# B&R Automation Studio project A2019059_Linka_Power_CP (part 60)

#### Main.st - Init, cyclic, exit code
```iecst
PROGRAM _INIT
	(* Insert code here *)

END_PROGRAM

PROGRAM _CYCLIC

	//Alarmy pracoviska č.1 (100 - 199)//
	//A100 - ST1_Vytah - paletka na vystupe dopravnika vytahu !!!
	//A101 - ST1_Vytah - narusenie optickej bariery !!!
	//A102 - ST1_Vytah - porucha navezenia paletky na dopravnik vytahu !!!
	//A103 - ST1_Vytah - porucha precitania kodu paletky !!!
	//A104 - ST1_Vytah - porucha komunikacie zo serverom !!!
	//A105 - ST1_Vytah - porucha odoslania fotiek na server !!!
	//A106 - ST1_Vytah - CAM 2 porucha komunikacie FTP !!!
	//A107 - ST1_Vytah - CAM 3 porucha komunikacie FTP !!!
	//A108 - ST1_Vytah - CAM 4 porucha komunikacie FTP !!!
	//A109 - ST1_Vytah - CAM 5 porucha komunikacie FTP !!!
	//A110 - ST1_Vytah - porucha serva zdvihu vytahu !!!
	//A111 - ST2_Srobovanie - porucha vysunutia centrovacky !!!
	//A112 - ST2_Srobovanie - porucha zasunutia centrovacky !!!
	//A113 - ST2_Srobovanie - porucha precitania kodu paletky !!!
	//A114 - ST2_Srobovanie - porucha komunikacie zo serverom !!!
	//A115 - ST2_Srobovanie - porucha odoslania fotiek na server !!!
	//A116 - ST2_Srobovanie - CAM 6 porucha komunikacie FTP !!!
	//A117 - ST2_Srobovanie - porucha serva manipulatora os X !!!
	//A118 - ST2_Srobovanie - porucha serva manipulatora os Y !!!
	//A119 - ST2_Srobovanie - skrutka K30 nieje pripravena !!!
	//A120 - ST2_Srobovanie - skrutka M5 nieje pripravena !!!
    //A121 - ST2_Srobovanie - skrutka M4 nieje pripravena !!!
    //A122 - P1_Robot - porucha napajania !!!
    //A123 - P1_Robot - nieje online !!!
    //A124 - Pracovisko 1 - Porucha tlaku vzduchu !!!
    //A125 - Pracovisko 1 - Modul DI11 nieje online !!!
    //A126 - Pracovisko 1 - Modul DI12 nieje online !!!
    //A127 - Pracovisko 1 - Modul DI13 nieje online !!!
    //A128 - Pracovisko 1 - Modul DI14 nieje online !!!
    //A129 - Pracovisko 1 - Modul DM11 nieje online !!!
    //A130 - Pracovisko 1 - Modul DS11 nieje online !!!
	//A131 - Pracovisko 1 - Modul DS12 nieje online !!!
	//A132 - Pracovisko 1 - Modul SI11 nieje online !!!
	//A133 - Pracovisko 1 - Modul SI12 nieje online !!!
    //A134 - Pracovisko 1 - Ventilovy termnal VT4 nieje online !!!
    //A135 - Pracovisko 1 - Ventilovy termnal VT5 nieje online !!!
    //A136 - ST2_Srobovanie - Skrutkovacka K30 nieje online !!!
    //A137 - ST2_Srobovanie - Skrutkovacka M5 nieje online !!!
    //A138 - ST2_Srobovanie - Skrutkovacka M4 nieje online !!!
    //A139 - Pracovisko 1 - Kamery KAM2, KAM4 a KAM6 niesu online !!!
    //A140 - Pracovisko 1 - Kamera KAM3 nieje online !!!
	//A141 - Pracovisko 1 - Kamera KAM5 nieje online !!!
    //A142 - ST2_Srobovanie - Porucha vysunutia skrutkovacky K30 !!!
    //A143 - ST2_Srobovanie - Porucha vysunutia skrutkovacky M5  !!!
    //A144 - ST2_Srobovanie - Porucha vysunutia skrutkovacky M4 !!!
	//A145 - P1_Robot - porucha !!!
    //A146 - ST2_Srobovanie - Presiahnuty cas skrutkovania skrutky K30 !!!
    //A147 - ST2_Srobovanie - Presiahnuty cas skrutkovania skrutky M5 !!!
    //A148 - ST2_Srobovanie - Presiahnuty cas skrutkovania skrutky M4 !!!
    //A149 - ST2_Srobovanie - Skrutkovacka K30 nieje READY !!!
    //A150 - ST2_Srobovanie - Skrutkovacka M5 nieje READY !!!
    //A151 - ST2_Srobovanie - Skrutkovacka M4 nieje READY !!!
    //A152 - Pracovisko 1 - Prekrocena teplota motora vrchneho dopravnika !!!
    //A153 - Pracovisko 1 - Prekrocena teplota motora spodneho dopravnika !!!
    //A154 - Pracovisko 1 - Narusenie optickej bariery na vstupe !!!
    //A155 - ST1_Vytah - Prekrocena teplota motora dopravnika !!!
    //A156 - Pracovisko 1 - Bolo stlacene tlacitko CS na ovladacom paneli !!!
    //A157 - Pracovisko 1 - Bolo stlacene tlacitko CS na rozvodnej skrini !!!
    //A158 - Pracovisko 1 - Bolo stlacene tlacitko CS robota !!!
    //A159 - P1_Robot - Porucha odobratia foamov z paletky !!!
    //A160 - P1_Robot - Porucha odobratia busbarov z paletky !!!
    //A161 - ST2_Srobovanie - Porucha vyvezenia paletky zo stopra !!!
    //A162 - P1_Akumulacny stoper - Porucha vyvezenia paletky zo stopra !!!
    //A163 - P1_Spodny stoper - Porucha vyvezenia paletky zo stopra !!!
    //A164 - ST1_Vytah - Porucha komunikacie s kamerou CAM 2 !!!
    //A165 - ST1_Vytah - Porucha komunikacie s kamerou CAM 5 !!!
    //A166 - ST1_Vytah - Porucha komunikacie s kamerou CAM 4 !!!
    //A167 - ST1_Vytah - Porucha komunikacie s kamerou CAM 3 !!!
    //A168 - ST2_Srobovanie - Porucha komunikacie s kamerou CAM 6 !!!

	//******************************Configurácia alarmov**************************************//
    MpAlarmXCore_1.Enable:= TRUE;
    MpAlarmXCore_1.MpLink:= ADR(gAlarmXCore);
    MpAlarmXCore_1();

    //*****************************Configurácia histórie alarmov*****************************//

    MpAlarmXHistory_1.Enable:= TRUE;
    MpAlarmXHistory_1.MpLink:= ADR(gAlarmXHistory);
    MpAlarmXHistory_1.DeviceName:= ADR('HDD_AlarmHistory');
    MpAlarmXHistory_1();

    //****************************Archivácia alarmov na disk PLC******************************//
    IF P1_AlarmyVizu.ArchivaciaAlarmov THEN
        MpAlarmXHistory_1.Export:= TRUE;
        P1_AlarmyVizu.ArchivaciaAlarmov:= FALSE;
    ELSIF P2_AlarmyVizu.ArchivaciaAlarmov THEN
        MpAlarmXHistory_1.Export:= TRUE;
        P2_AlarmyVizu.ArchivaciaAlarmov:= FALSE;
    ELSIF P34_AlarmyVizu.ArchivaciaAlarmov THEN
        MpAlarmXHistory_1.Export:= TRUE;
        P34_AlarmyVizu.ArchivaciaAlarmov:= FALSE;
    END_IF

    IF MpAlarmXHistory_1.Error THEN
        MpAlarmXHistory_1.Export:= FALSE;
    ELSIF MpAlarmXHistory_1.CommandDone THEN
        MpAlarmXHistory_1.Export:= FALSE;
    END_IF

    //***********************************Príznak pracovisko 1 stav PORUCHA*****************************************//

    FOR a:=100 TO 199 BY 1 DO
        P1_Alarmy[a];
        IF P1_Alarmy[a] = TRUE THEN
            P1_Pracovisko.STAV.PORUCHA:= TRUE;
        END_IF
    END_FOR

    //**********************************Porucha tlaku vzduchu*********************************************************//
    IF CasKontroly_TlakVzduchu.Q THEN
        P1_Alarmy[124]:= TRUE;
        P1_PoruchaST1:= TRUE;
        P1_PoruchaST2:= TRUE;
    END_IF

    IF Safety.STAV.P1_ZonaBunky_AKTIVNA AND NOT P1_Pracovisko.IN.PrivodVzduchu_SnimacTlaku_S18 THEN
        CasKontroly_TlakVzduchu.IN:= TRUE;
    ELSE
        CasKontroly_TlakVzduchu.IN:= FALSE;
    END_IF

    CasKontroly_TlakVzduchu.PT:= T#10s;
    CasKontroly_TlakVzduchu();

    //**********************************Porucha - kamerovy systém nieje online****************************************//
    IF CasKontroly_KAMsystem.Q THEN
        IF NOT Linka.STAV.WenglorControlUnit_OK THEN
            P1_Alarmy[149]:= TRUE;
            P1_PoruchaST1:= TRUE;
            P1_PoruchaST2:= TRUE;
        END_IF
        IF NOT CAM3.STAV.READY THEN
            P1_Alarmy[140]:= TRUE;
            P1_PoruchaST1:= TRUE;
            P1_PoruchaST2:= TRUE;
        END_IF
        IF NOT CAM5.STAV.READY THEN
            P1_Alarmy[141]:= TRUE;
            P1_PoruchaST1:= TRUE;
            P1_PoruchaST2:= TRUE;
        END_IF
    END_IF

    IF Safety.STAV.P1_ZonaBunky_AKTIVNA AND NOT P1_Pracovisko.STAV.Kamery_OK THEN
        CasKontroly_KAMsystem.IN:= TRUE;
    ELSE
        CasKontroly_KAMsystem.IN:= FALSE;
    END_IF

    CasKontroly_KAMsystem.PT:= T#2s;
    CasKontroly_KAMsystem();

    //**********************************Porucha - moduly niesu online**************************************************//
    IF CasKontroly_Moduly.Q THEN
        IF NOT P1_Pracovisko.STAV.ModulDI11_OK THEN
            P1_Alarmy[125]:= TRUE;
            P1_PoruchaST1:= TRUE;
            P1_PoruchaST2:= TRUE;
        END_IF
        IF NOT P1_Pracovisko.STAV.ModulDI12_OK THEN
            P1_Alarmy[126]:= TRUE;
            P1_PoruchaST1:= TRUE;
            P1_PoruchaST2:= TRUE;
        END_IF
        IF NOT P1_Pracovisko.STAV.ModulDI13_OK THEN
            P1_Alarmy[127]:= TRUE;
            P1_PoruchaST1:= TRUE;
            P1_PoruchaST2:= TRUE;
        END_IF
        IF NOT P1_Pracovisko.STAV.ModulDI14_OK THEN
            P1_Alarmy[128]:= TRUE;
            P1_PoruchaST1:= TRUE;
            P1_PoruchaST2:= TRUE;
        END_IF
        IF NOT P1_Pracovisko.STAV.ModulDM11_OK THEN
            P1_Alarmy[129]:= TRUE;
            P1_PoruchaST1:= TRUE;
            P1_PoruchaST2:= TRUE;
        END_IF
        IF NOT P1_Pracovisko.STAV.ModulDS11_OK THEN
            P1_Alarmy[130]:= TRUE;
            P1_PoruchaST1:= TRUE;
            P1_PoruchaST2:= TRUE;
        END_IF
        IF NOT P1_Pracovisko.STAV.ModulDS12_OK THEN
            P1_Alarmy[131]:= TRUE;
            P1_PoruchaST1:= TRUE;
            P1_PoruchaST2:= TRUE;
        END_IF
        IF NOT P1_Pracovisko.STAV.ModulSI11_OK THEN
            P1_Alarmy[132]:= TRUE;
            P1_PoruchaST1:= TRUE;
            P1_PoruchaST2:= TRUE;
        END_IF
        IF NOT P1_Pracovisko.STAV.ModulSI12_OK THEN
            P1_Alarmy[133]:= TRUE;
            P1_PoruchaST1:= TRUE;
            P1_PoruchaST2:= TRUE;
        END_IF
    END_IF

    IF Safety.STAV.P1_ZonaBunky_AKTIVNA AND NOT P1_Pracovisko.STAV.Moduly_OK THEN
        CasKontroly_Moduly.IN:= TRUE;
    ELSE
        CasKontroly_Moduly.IN:= FALSE;
    END_IF

    CasKontroly_Moduly.PT:= T#2s;
    CasKontroly_Moduly();

    //********************************Porucha - ventilové terminály niesu online**********************************************//
    IF CasKontroly_VentTerminalov.Q THEN
        IF NOT P1_Pracovisko.STAV.VentilovyTerminal_VT4_OK THEN
            P1_Alarmy[134]:= TRUE;
            P1_PoruchaST1:= TRUE;
            P1_PoruchaST2:= TRUE;
        END_IF
        IF NOT P1_Pracovisko.STAV.VentilovyTerminal_VT5_OK THEN
            P1_Alarmy[135]:= TRUE;
            P1_PoruchaST1:= TRUE;
            P1_PoruchaST2:= TRUE;
        END_IF
    END_IF

    IF Safety.STAV.P1_ZonaBunky_AKTIVNA AND NOT P1_Pracovisko.STAV.VentiloveTerminaly_OK THEN
        CasKontroly_VentTerminalov.IN:= TRUE;
    ELSE
        CasKontroly_VentTerminalov.IN:= FALSE;
    END_IF

    CasKontroly_VentTerminalov.PT:= T#2s;
    CasKontroly_VentTerminalov();

    //********************************Porucha - skrutkovacky niesu online**********************************************//
    IF CasKontroly_Skrutkovacky.Q THEN
        IF NOT P1_Pracovisko.STAV.Skrutkovacka_K30_OK THEN
            P1_Alarmy[136]:= TRUE;
            P1_PoruchaST2:= TRUE;
        END_IF
        IF NOT P1_Pracovisko.STAV.Skrutkovacka_M5_OK THEN
            P1_Alarmy[137]:= TRUE;
            P1_PoruchaST2:= TRUE;
        END_IF
        IF NOT P1_Pracovisko.STAV.Skrutkovacka_M4_OK THEN
            P1_Alarmy[138]:= TRUE;
            P1_PoruchaST2:= TRUE;
        END_IF
    END_IF

    IF Safety.STAV.P1_ZonaBunky_AKTIVNA AND NOT P1_Pracovisko.STAV.Skrutkovacky_OK THEN
        CasKontroly_Skrutkovacky.IN:= TRUE;
    ELSE
        CasKontroly_Skrutkovacky.IN:= FALSE;
    END_IF

    CasKontroly_Skrutkovacky.PT:= T#2s;
    CasKontroly_Skrutkovacky();

    //*********************************Porucha - robot nieje online************************************************//
    IF CasKontroly_Robota.Q THEN
        P1_Alarmy[123]:= TRUE;
        P1_PoruchaST2:= TRUE;
    END_IF

    IF Safety.STAV.P1_ZonaBunky_AKTIVNA AND NOT P1_Pracovisko.STAV.KOM_Robot_OK THEN
        CasKontroly_Robota.IN:= TRUE;
    ELSE
        CasKontroly_Robota.IN:= FALSE;
    END_IF

    CasKontroly_Robota.PT:= T#2s;
    CasKontroly_Robota();

    //*******************************Porucha napájania robota*****************************************************//
    IF CasKontroly_Robota.Q AND NOT P1_Pracovisko.IN.NapajaniaRobota_OK THEN
        P1_Alarmy[122]:= TRUE;
        P1_PoruchaST2:= TRUE;
    END_IF

    //********************Pracovisko 1 - Porucha ochrannej bariéry výťahu****************************************//

    IF Safety.IN.P1_Vytah_Zdvih_BUSY AND NOT Safety.STAV.P1_Vytah_Bariera_AKTIVNA THEN
        P1_Alarmy[101]:= TRUE;
        P1_PoruchaST1:= TRUE;
    END_IF

    IF Safety.IN.P1_Vytah_Zdvih_BUSY AND P1_Vytah.IN.VystupDopravnikaVytahu_OS12 THEN
        P1_Alarmy[101]:= TRUE;
        P1_PoruchaST1:= TRUE;
    END_IF

    //*********************Pracovisko 1 - Porucha serva zdvihu vytahu***************//
    IF CasPoruchyServaVytahu.Q THEN
        P1_Alarmy[110]:= TRUE;
        P1_PoruchaST1:= TRUE;
    END_IF

    IF Safety.STAV.P1_ZonaVytahu_AKTIVNA AND P1_Vytah.ServoZdvihuVytahu_M31.STATUS.ERROR THEN
        CasPoruchyServaVytahu.IN:= TRUE;
    ELSE
        CasPoruchyServaVytahu.IN:= FALSE;
    END_IF

    CasPoruchyServaVytahu.PT:= T#2s;
    CasPoruchyServaVytahu();

    //*********************Pracovisko 1 - Porucha serva manipulatora šrobovania os X***************//
    IF CasPoruchyServaSrobovaniaOsX.Q THEN
        P1_Alarmy[117]:= TRUE;
        P1_PoruchaST2:= TRUE;
    END_IF

    IF Safety.STAV.P1_ZonaBunky_AKTIVNA AND P1_Srobovanie.ServoManipulOsX_M20.STATUS.ERROR THEN
        CasPoruchyServaSrobovaniaOsX.IN:= TRUE;
    ELSE
        CasPoruchyServaSrobovaniaOsX.IN:= FALSE;
    END_IF

    CasPoruchyServaSrobovaniaOsX.PT:= T#2s;
    CasPoruchyServaSrobovaniaOsX();

    //*********************Pracovisko 1 - Porucha serva manipulatora šrobovania os Y***************//
    IF CasPoruchyServaSrobovaniaOsY.Q THEN
        P1_Alarmy[118]:= TRUE;
        P1_PoruchaST2:= TRUE;
    END_IF

    IF Safety.STAV.P1_ZonaBunky_AKTIVNA AND P1_Srobovanie.ServoManipulOsY_M19.STATUS.ERROR THEN
        CasPoruchyServaSrobovaniaOsY.IN:= TRUE;
    ELSE
        CasPoruchyServaSrobovaniaOsY.IN:= FALSE;
    END_IF

    CasPoruchyServaSrobovaniaOsY.PT:= T#2s;
    CasPoruchyServaSrobovaniaOsY();

    //****************************Pracovisko 1 - porucha vrchného dopravníka**********************************//
    IF NOT P1_Dopravniky.IN.HornyDoprav_TeplotaMotora_OK AND P1_Pracovisko.STAV.Automat THEN
        P1_Alarmy[152]:= TRUE;
    END_IF

    //*****************************Pracovisko 1 - porucha spodného dopravníka************************************//
    IF NOT P1_Dopravniky.IN.SpodnyDoprav_TeplotaMotora_OK AND P1_Pracovisko.STAV.Automat THEN
        P1_Alarmy[153]:= TRUE;
    END_IF

    //******************************Pracovisko 1 - narušenie vstupnej bariery***********************************//
    IF NOT Safety.STAV.P1_VstupBunky_Bariera_AKTIVNA AND NOT Safety.STAV.P1_VystupTunela_Bariera_AKTIVNA AND P1_Pracovisko.STAV.Automat THEN
        P1_Alarmy[154]:= TRUE;
    END_IF

    //******************************Výťah - porucha dopravníka**************************************************//
    IF NOT P1_Vytah.IN.Dopravnik_TeplotaMotora_OK AND P1_Vytah.Automat THEN
        P1_Alarmy[155]:= TRUE;
        P1_PoruchaST1:= TRUE;
    END_IF

    //******************************Stlačenie tlačítok CS*******************************************************//
    IF EDGENEG(Safety.STAV.P1_Panel_TlacitkoCS_AKTIVNE) THEN
        P1_Alarmy[156]:= TRUE;
    END_IF

    IF EDGENEG(Safety.STAV.P1_Skrina_TlacitkoCS_AKTIVNE) THEN
        P1_Alarmy[157]:= TRUE;
    END_IF

    IF EDGENEG(Safety.STAV.P1_Robot_TlacitkoCS_AKTIVNE) THEN
        P1_Alarmy[158]:= TRUE;
    END_IF

    //***************************************************Nasetovanie alarmov****************************************************//
    IF P1_Alarmy[100] THEN
        MpAlarmXSet(gAlarmXCore, 'A100');
    ELSE
        MpAlarmXReset(gAlarmXCore, 'A100');
    END_IF

    IF P1_Alarmy[101] THEN
        MpAlarmXSet(gAlarmXCore, 'A101');
    ELSE
        MpAlarmXReset(gAlarmXCore, 'A101');
    END_IF

    IF P1_Alarmy[102] THEN
        MpAlarmXSet(gAlarmXCore, 'A102');
    ELSE
        MpAlarmXReset(gAlarmXCore, 'A102');
    END_IF

    IF P1_Alarmy[103] THEN
        MpAlarmXSet(gAlarmXCore, 'A103');
    ELSE
        MpAlarmXReset(gAlarmXCore, 'A103');
    END_IF

    IF P1_Alarmy[104] THEN
        MpAlarmXSet(gAlarmXCore, 'A104');
    ELSE
        MpAlarmXReset(gAlarmXCore, 'A104');
    END_IF

    IF P1_Alarmy[105] THEN
        MpAlarmXSet(gAlarmXCore, 'A105');
    ELSE
        MpAlarmXReset(gAlarmXCore, 'A105');
    END_IF

    IF P1_Alarmy[106] THEN
        MpAlarmXSet(gAlarmXCore, 'A106');
    ELSE
        MpAlarmXReset(gAlarmXCore, 'A106');
    END_IF

    IF P1_Alarmy[107] THEN
        MpAlarmXSet(gAlarmXCore, 'A107');
    ELSE
        MpAlarmXReset(gAlarmXCore, 'A107');
    END_IF

    IF P1_Alarmy[108] THEN
        MpAlarmXSet(gAlarmXCore, 'A108');
    ELSE
        MpAlarmXReset(gAlarmXCore, 'A108');
    END_IF

    IF P1_Alarmy[109] THEN
        MpAlarmXSet(gAlarmXCore, 'A109');
    ELSE
        MpAlarmXReset(gAlarmXCore, 'A109');
    END_IF

    IF P1_Alarmy[110] THEN
        MpAlarmXSet(gAlarmXCore, 'A110');
    ELSE
        MpAlarmXReset(gAlarmXCore, 'A110');
    END_IF

    IF P1_Alarmy[111] THEN
        MpAlarmXSet(gAlarmXCore, 'A111');
    ELSE
        MpAlarmXReset(gAlarmXCore, 'A111');
    END_IF

    IF P1_Alarmy[112] THEN
        MpAlarmXSet(gAlarmXCore, 'A112');
    ELSE
        MpAlarmXReset(gAlarmXCore, 'A112');
    END_IF

    IF P1_Alarmy[113] THEN
        MpAlarmXSet(gAlarmXCore, 'A113');
    ELSE
        MpAlarmXReset(gAlarmXCore, 'A113');
    END_IF

    IF P1_Alarmy[114] THEN
        MpAlarmXSet(gAlarmXCore, 'A114');
    ELSE
        MpAlarmXReset(gAlarmXCore, 'A114');
    END_IF

    IF P1_Alarmy[115] THEN
        MpAlarmXSet(gAlarmXCore, 'A115');
    ELSE
        MpAlarmXReset(gAlarmXCore, 'A115');
    END_IF

    IF P1_Alarmy[116] THEN
        MpAlarmXSet(gAlarmXCore, 'A116');
    ELSE
        MpAlarmXReset(gAlarmXCore, 'A116');
    END_IF

    IF P1_Alarmy[117] THEN
        MpAlarmXSet(gAlarmXCore, 'A117');
    ELSE
        MpAlarmXReset(gAlarmXCore, 'A117');
    END_IF

    IF P1_Alarmy[118] THEN
        MpAlarmXSet(gAlarmXCore, 'A118');
    ELSE
        MpAlarmXReset(gAlarmXCore, 'A118');
    END_IF

    IF P1_Alarmy[119] THEN
        MpAlarmXSet(gAlarmXCore, 'A119');
    ELSE
        MpAlarmXReset(gAlarmXCore, 'A119');
    END_IF

    IF P1_Alarmy[120] THEN
        MpAlarmXSet(gAlarmXCore, 'A120');
    ELSE
        MpAlarmXReset(gAlarmXCore, 'A120');
    END_IF

    IF P1_Alarmy[121] THEN
        MpAlarmXSet(gAlarmXCore, 'A121');
    ELSE
        MpAlarmXReset(gAlarmXCore, 'A121');
    END_IF

    IF P1_Alarmy[122] THEN
        MpAlarmXSet(gAlarmXCore, 'A122');
    ELSE
        MpAlarmXReset(gAlarmXCore, 'A122');
    END_IF

    IF P1_Alarmy[123] THEN
        MpAlarmXSet(gAlarmXCore, 'A123');
    ELSE
        MpAlarmXReset(gAlarmXCore, 'A123');
    END_IF

    IF P1_Alarmy[124] THEN
        MpAlarmXSet(gAlarmXCore, 'A124');
    ELSE
        MpAlarmXReset(gAlarmXCore, 'A124');
    END_IF

    IF P1_Alarmy[125] THEN
        MpAlarmXSet(gAlarmXCore, 'A125');
    ELSE
        MpAlarmXReset(gAlarmXCore, 'A125');
    END_IF

    IF P1_Alarmy[126] THEN
        MpAlarmXSet(gAlarmXCore, 'A126');
    ELSE
        MpAlarmXReset(gAlarmXCore, 'A126');
    END_IF

    IF P1_Alarmy[127] THEN
        MpAlarmXSet(gAlarmXCore, 'A127');
    ELSE
        MpAlarmXReset(gAlarmXCore, 'A127');
    END_IF

    IF P1_Alarmy[128] THEN
        MpAlarmXSet(gAlarmXCore, 'A128');
    ELSE
        MpAlarmXReset(gAlarmXCore, 'A128');
    END_IF

    IF P1_Alarmy[129] THEN
        MpAlarmXSet(gAlarmXCore, 'A129');
    ELSE
        MpAlarmXReset(gAlarmXCore, 'A129');
    END_IF

    IF P1_Alarmy[130] THEN
        MpAlarmXSet(gAlarmXCore, 'A130');
    ELSE
        MpAlarmXReset(gAlarmXCore, 'A130');
    END_IF

    IF P1_Alarmy[131] THEN
        MpAlarmXSet(gAlarmXCore, 'A131');
    ELSE
        MpAlarmXReset(gAlarmXCore, 'A131');
    END_IF

    IF P1_Alarmy[132] THEN
        MpAlarmXSet(gAlarmXCore, 'A132');
    ELSE
        MpAlarmXReset(gAlarmXCore, 'A132');
    END_IF

    IF P1_Alarmy[133] THEN
        MpAlarmXSet(gAlarmXCore, 'A133');
    ELSE
        MpAlarmXReset(gAlarmXCore, 'A133');
    END_IF

    IF P1_Alarmy[134] THEN
        MpAlarmXSet(gAlarmXCore, 'A134');
    ELSE
        MpAlarmXReset(gAlarmXCore, 'A134');
    END_IF

    IF P1_Alarmy[135] THEN
        MpAlarmXSet(gAlarmXCore, 'A135');
    ELSE
        MpAlarmXReset(gAlarmXCore, 'A135');
    END_IF

    IF P1_Alarmy[136] THEN
        MpAlarmXSet(gAlarmXCore, 'A136');
    ELSE
        MpAlarmXReset(gAlarmXCore, 'A136');
    END_IF

    IF P1_Alarmy[137] THEN
        MpAlarmXSet(gAlarmXCore, 'A137');
    ELSE
        MpAlarmXReset(gAlarmXCore, 'A137');
    END_IF

    IF P1_Alarmy[138] THEN
        MpAlarmXSet(gAlarmXCore, 'A138');
    ELSE
        MpAlarmXReset(gAlarmXCore, 'A138');
    END_IF

    IF P1_Alarmy[139] THEN
        MpAlarmXSet(gAlarmXCore, 'A139');
    ELSE
        MpAlarmXReset(gAlarmXCore, 'A139');
    END_IF

    IF P1_Alarmy[140] THEN
        MpAlarmXSet(gAlarmXCore, 'A140');
    ELSE
        MpAlarmXReset(gAlarmXCore, 'A140');
    END_IF

    IF P1_Alarmy[141] THEN
        MpAlarmXSet(gAlarmXCore, 'A141');
    ELSE
        MpAlarmXReset(gAlarmXCore, 'A141');
    END_IF

    IF P1_Alarmy[142] THEN
        MpAlarmXSet(gAlarmXCore, 'A142');
    ELSE
        MpAlarmXReset(gAlarmXCore, 'A142');
    END_IF

    IF P1_Alarmy[143] THEN
        MpAlarmXSet(gAlarmXCore, 'A143');
    ELSE
        MpAlarmXReset(gAlarmXCore, 'A143');
    END_IF

    IF P1_Alarmy[144] THEN
        MpAlarmXSet(gAlarmXCore, 'A144');
    ELSE
        MpAlarmXReset(gAlarmXCore, 'A144');
    END_IF

    IF P1_Alarmy[145] THEN
        MpAlarmXSet(gAlarmXCore, 'A145');
    ELSE
        MpAlarmXReset(gAlarmXCore, 'A145');
    END_IF

    IF P1_Alarmy[146] THEN
        MpAlarmXSet(gAlarmXCore, 'A146');
    ELSE
        MpAlarmXReset(gAlarmXCore, 'A146');
    END_IF

    IF P1_Alarmy[147] THEN
        MpAlarmXSet(gAlarmXCore, 'A147');
    ELSE
        MpAlarmXReset(gAlarmXCore, 'A147');
    END_IF

    IF P1_Alarmy[148] THEN
        MpAlarmXSet(gAlarmXCore, 'A148');
    ELSE
        MpAlarmXReset(gAlarmXCore, 'A148');
    END_IF

    IF P1_Alarmy[149] THEN
        MpAlarmXSet(gAlarmXCore, 'A149');
    ELSE
        MpAlarmXReset(gAlarmXCore, 'A149');
    END_IF

    IF P1_Alarmy[150] THEN
        MpAlarmXSet(gAlarmXCore, 'A150');
    ELSE
        MpAlarmXReset(gAlarmXCore, 'A150');
    END_IF

    IF P1_Alarmy[151] THEN
        MpAlarmXSet(gAlarmXCore, 'A151');
    ELSE
        MpAlarmXReset(gAlarmXCore, 'A151');
    END_IF

    IF P1_Alarmy[152] THEN
        MpAlarmXSet(gAlarmXCore, 'A152');
    ELSE
        MpAlarmXReset(gAlarmXCore, 'A152');
    END_IF

    IF P1_Alarmy[153] THEN
        MpAlarmXSet(gAlarmXCore, 'A153');
    ELSE
        MpAlarmXReset(gAlarmXCore, 'A153');
    END_IF

    IF P1_Alarmy[154] THEN
        MpAlarmXSet(gAlarmXCore, 'A154');
    ELSE
        MpAlarmXReset(gAlarmXCore, 'A154');
    END_IF

    IF P1_Alarmy[155] THEN
        MpAlarmXSet(gAlarmXCore, 'A155');
    ELSE
        MpAlarmXReset(gAlarmXCore, 'A155');
    END_IF

    IF P1_Alarmy[156] THEN
        MpAlarmXSet(gAlarmXCore, 'A156');
    ELSE
        MpAlarmXReset(gAlarmXCore, 'A156');
    END_IF

    IF P1_Alarmy[157] THEN
        MpAlarmXSet(gAlarmXCore, 'A157');
    ELSE
        MpAlarmXReset(gAlarmXCore, 'A157');
    END_IF

    IF P1_Alarmy[158] THEN
        MpAlarmXSet(gAlarmXCore, 'A158');
    ELSE
        MpAlarmXReset(gAlarmXCore, 'A158');
    END_IF

    IF P1_Alarmy[159] THEN
        MpAlarmXSet(gAlarmXCore, 'A159');
    ELSE
        MpAlarmXReset(gAlarmXCore, 'A159');
    END_IF

    IF P1_Alarmy[160] THEN
        MpAlarmXSet(gAlarmXCore, 'A160');
    ELSE
        MpAlarmXReset(gAlarmXCore, 'A160');
    END_IF

    IF P1_Alarmy[161] THEN
        MpAlarmXSet(gAlarmXCore, 'A161');
    ELSE
        MpAlarmXReset(gAlarmXCore, 'A161');
    END_IF

    IF P1_Alarmy[162] THEN
        MpAlarmXSet(gAlarmXCore, 'A162');
    ELSE
        MpAlarmXReset(gAlarmXCore, 'A162');
    END_IF

    IF P1_Alarmy[163] THEN
        MpAlarmXSet(gAlarmXCore, 'A163');
    ELSE
        MpAlarmXReset(gAlarmXCore, 'A163');
    END_IF

    IF P1_Alarmy[164] THEN
        MpAlarmXSet(gAlarmXCore, 'A164');
    ELSE
        MpAlarmXReset(gAlarmXCore, 'A164');
    END_IF

    IF P1_Alarmy[165] THEN
        MpAlarmXSet(gAlarmXCore, 'A165');
    ELSE
        MpAlarmXReset(gAlarmXCore, 'A165');
    END_IF

    IF P1_Alarmy[166] THEN
        MpAlarmXSet(gAlarmXCore, 'A166');
    ELSE
        MpAlarmXReset(gAlarmXCore, 'A166');
    END_IF

    IF P1_Alarmy[167] THEN
        MpAlarmXSet(gAlarmXCore, 'A167');
    ELSE
        MpAlarmXReset(gAlarmXCore, 'A167');
    END_IF

    IF P1_Alarmy[168] THEN
        MpAlarmXSet(gAlarmXCore, 'A168');
    ELSE
        MpAlarmXReset(gAlarmXCore, 'A168');
    END_IF

    //********************************Zobrazenie symbolu alarmu*****************************************************//

    IF P1_Pracovisko.STAV.PORUCHA THEN
        P1_AlarmyVizu.ZobrazSymbolAlarmu:= Blikac500ms;
    ELSE
        P1_AlarmyVizu.ZobrazSymbolAlarmu:= FALSE;
    END_IF

    //********************************Blikanie tlačítka Alarmy*******************************************************//
    IF P1_Pracovisko.STAV.PORUCHA AND P1_Vizu.ActualPage <> 'PageAlarm' THEN
        IF Blikac500ms THEN
            P1_AlarmyVizu.FarbaTlacitka_Alarmy:= "Button_Red";
        ELSE
            P1_AlarmyVizu.FarbaTlacitka_Alarmy:= "default";
        END_IF
    ELSE
        P1_AlarmyVizu.FarbaTlacitka_Alarmy:= "default";
    END_IF

    //*************************************Potvrdenie alarmov*********************************************************//
    IF P1_AlarmyVizu.PotvrdAlarmy THEN
        brsmemset(ADR(P1_Alarmy),0,SIZEOF(P1_Alarmy));
        P1_Pracovisko.STAV.PORUCHA:= FALSE;
        P1_PoruchaST1:= FALSE;
        P1_PoruchaST2:= FALSE;
        IF P1_Vytah.ServoZdvihuVytahu_M31.STATUS.ERROR AND P1_Vytah.ServoZdvihuVytahu_M31.STATUS.ReadyToPower_ON THEN
            P1_Vytah.ServoZdvihuVytahu_M31.CMD.ErrorRESET:= TRUE;
        END_IF
        IF P1_Srobovanie.ServoManipulOsX_M20.STATUS.ERROR AND P1_Srobovanie.ServoManipulOsX_M20.STATUS.ReadyToPower_ON THEN
            P1_Srobovanie.ServoManipulOsX_M20.CMD.ErrorRESET:= TRUE;
        END_IF
        IF P1_Srobovanie.ServoManipulOsY_M19.STATUS.ERROR AND P1_Srobovanie.ServoManipulOsY_M19.STATUS.ReadyToPower_ON THEN
            P1_Srobovanie.ServoManipulOsY_M19.CMD.ErrorRESET:= TRUE;
        END_IF
        P1_AlarmyVizu.PotvrdAlarmy:= FALSE;
    END_IF

    //Resetovanie serva zdvihu výťahu//
    IF EDGEPOS(Safety.STAV.P1_ZonaVytahu_AKTIVNA) THEN
        P1_Vytah.ServoZdvihuVytahu_M31.CMD.ErrorRESET:= TRUE;
    END_IF

    //Resetovanie poruch serv pri zatvorení bunky//
    IF EDGEPOS(Safety.STAV.P1_ZonaBunky_AKTIVNA) THEN
        P1_Srobovanie.ServoManipulOsX_M20.CMD.ErrorRESET:= TRUE;
        P1_Srobovanie.ServoManipulOsY_M19.CMD.ErrorRESET:= TRUE;
    END_IF

    //Zrušenie resetovania porúch serv//
    IF NOT P1_Vytah.ServoZdvihuVytahu_M31.STATUS.ERROR THEN
        P1_Vytah.ServoZdvihuVytahu_M31.CMD.ErrorRESET:= FALSE;
    ELSIF CasResetovaniaServaZdvihuVytahu.Q THEN
        P1_Vytah.ServoZdvihuVytahu_M31.CMD.ErrorRESET:= FALSE;
    END_IF

    IF NOT P1_Srobovanie.ServoManipulOsX_M20.STATUS.ERROR THEN
        P1_Srobovanie.ServoManipulOsX_M20.CMD.ErrorRESET:= FALSE;
    ELSIF CasResetovaniaServaSrobovaniaOsX.Q THEN
        P1_Srobovanie.ServoManipulOsX_M20.CMD.ErrorRESET:= FALSE;
    END_IF

    IF NOT P1_Srobovanie.ServoManipulOsY_M19.STATUS.ERROR THEN
        P1_Srobovanie.ServoManipulOsY_M19.CMD.ErrorRESET:= FALSE;
    ELSIF CasResetovaniaServaSrobovaniaOsY.Q THEN
        P1_Srobovanie.ServoManipulOsY_M19.CMD.ErrorRESET:= FALSE;
    END_IF

    CasResetovaniaServaZdvihuVytahu.PT:= T#2s;
    CasResetovaniaServaZdvihuVytahu.IN:= P1_Vytah.ServoZdvihuVytahu_M31.CMD.ErrorRESET;
    CasResetovaniaServaZdvihuVytahu();

    CasResetovaniaServaSrobovaniaOsX.PT:= T#2s;
    CasResetovaniaServaSrobovaniaOsX.IN:= P1_Srobovanie.ServoManipulOsX_M20.CMD.ErrorRESET;
    CasResetovaniaServaSrobovaniaOsX();

    CasResetovaniaServaSrobovaniaOsY.PT:= T#2s;
    CasResetovaniaServaSrobovaniaOsY.IN:= P1_Srobovanie.ServoManipulOsY_M19.CMD.ErrorRESET;
    CasResetovaniaServaSrobovaniaOsY();

        END_PROGRAM

PROGRAM _EXIT
        (* Insert code here *)

        END_PROGRAM
```

#### Variables.var - Local variables
```iecst
VAR
	i : UINT;
	CasKontroly_KAMsystem : TON;
	CasKontroly_TlakVzduchu : TON;
	CasKontroly_Moduly : TON;
	CasKontroly_Robota : TON;
	CasKontroly_VentTerminalov : TON;
	CasKontroly_Skrutkovacky : TON;
	CasPoruchyServaVytahu : TON;
	CasPoruchyServaSrobovaniaOsY : TON;
	CasPoruchyServaSrobovaniaOsX : TON;
	CasResetovaniaServaZdvihuVytahu : TON;
	CasResetovaniaServaSrobovaniaOsX : TON;
	CasResetovaniaServaSrobovaniaOsY : TON;
	a : INT;
END_VAR
```

### Program Logical/Alarmy/P2_Alarmy (IEC)

#### Main.st - Init, cyclic, exit code
```iecst
PROGRAM _INIT
	(* Insert code here *)

END_PROGRAM

PROGRAM _CYCLIC

	//Alarmy pracoviska č.2 (200 - 299)//
	//A200 - ST3_Zakladanie tesnenia - porucha precitania kodu paletky !!!
	//A201 - ST3_Zakladanie tesnenia - porucha precitania QR kodu !!!
	//A202 - ST3_Zakladanie tesnenia - porucha serva zdvihu !!!
	//A203 - ST3_Zakladanie tesnenia - porucha serva pojazdu !!!
	//A204 - ST3_Zakladanie tesnenia - porucha vysunutia pritlacania !!!
	//A205 - ST3_Zakladanie tesnenia - porucha zasunutia pritlacania !!!
	//A206 - ST3_Zakladanie tesnenia - narusenie optickej bariery !!!
	//A207 - ST3_Zakladanie tesnenia - bol stlaceny bumper suflika !!!
	//A208 - ST3_Zakladanie tesnenia - porucha snimaca kopita IS7 !!!
	//A209 - ST4_Maticovacka - porucha vysunutia centrovacky !!!
	//A210 - ST4_Maticovacka - porucha zasunutia centrovacky !!!
	//A211 - ST4_Maticovacka - porucha precitania kodu paletky !!!
	//A212 - ST5_Srobovanie - porucha vysunutia centrovacky !!!
	//A213 - ST5_Srobovanie - porucha zasunutia centrovacky !!!
	//A214 - ST5_Srobovanie - porucha precitania kodu paletky !!!
	//A215 - ST5_Srobovanie - porucha serva manipulatora os X !!!
	//A216 - ST5_Srobovanie - porucha serva manipulatora os Y !!!
	//A217 - ST6_Zvaranie - porucha vysunutia centrovacky !!!
	//A218 - ST6_Zvaranie - porucha zasunutia centrovacky !!!
	//A219 - ST6_Zvaranie - porucha precitania kodu paletky !!!
	//A220 - ST6_Zvaranie - porucha serva zdvihu zvarania !!!
	//A221 - ST6_Zvaranie - porucha presunu pojazdu zvarania !!!
	//A222 - ST6_Zvaranie - porucha zvaracky !!!
	//A223 - ST6_Cistenie - porucha zatvorenia dveri !!!
	//A224 - ST6_Cistenie - porucha otvorenia dveri !!!
	//A225 - ST3_Zakladanie tesnenia - CAM 1 porucha komunikacie FTP !!!
	//A226 - ST3_Zakladanie tesnenia - CAM 7 porucha komunikacie FTP !!!
	//A227 - ST3_Zakladanie tesnenia - CAM 8 porucha komunikacie FTP !!!
	//A228 - ST3_Zakladanie tesnenia - CAM 17 porucha komunikacie FTP !!!
	//A229 - ST4_Maticovacka - CAM 9 porucha komunikacie FTP !!!
	//A230 - ST3_Zakladanie tesnenia - porucha komunikacie zo serverom !!!
	//A231 - ST4_Maticovacka - porucha komunikacie zo serverom !!!
	//A232 - ST5_Srobovanie - CAM 10 porucha komunikacie FTP !!!
	//A233 - ST5_Srobovanie - porucha komunikacie zo serverom !!!
	//A234 - ST6_Zvaranie - CAM 11 porucha komunikacie FTP !!!
	//A235 - ST6_Zvaranie - CAM 12 porucha komunikacie FTP !!!
	//A236 - ST6_Zvaranie - porucha komunikacie zo serverom !!!
	//A237 - ST5_Srobovanie - skrutka M4 nieje pripravena !!!
	//A238 - ST5_Srobovanie - skrutka M5 nieje pripravena !!!
	//A239 - ST5_Srobovanie - skrutka M6 nieje pripravena !!!
	//A240 - ST4_Maticovacka - matica M4 nieje pripravena !!!
	//A241 - ST5_Srobovanie - porucha serva manipulatora os X !!!
	//A242 - ST5_Srobovanie - porucha serva manipulatora os Y !!!
	//A243 - P2_Robot - porucha napajania !!!
	//A244 - P2_Robot - nieje online !!!
	//A245 - Pracovisko 2 - Porucha tlaku vzduchu !!!
	//A246 - Pracovisko 2 - Modul DI21 nieje online !!!
	//A247 - Pracovisko 2 - Modul DI22 nieje online !!!
	//A248 - Pracovisko 2 - Modul DI23 nieje online !!!
	//A249 - Pracovisko 2 - Modul DI24 nieje online !!!
	//A250 - Pracovisko 2 - Modul DI25 nieje online !!!
	//A251 - Pracovisko 2 - Modul DM21 nieje online !!!
	//A252 - Pracovisko 2 - Modul DS21 nieje online !!!
    //A253 - Pracovisko 2 - Modul DS22 nieje online !!!
    //A254 - Pracovisko 2 - Modul DS23 nieje online !!!
	//A255 - Pracovisko 2 - Modul SI21 nieje online !!!
    //A256 - Pracovisko 2 - Modul SI22 nieje online !!!
	//A257 - Pracovisko 2 - Ventilovy termnal VT1 nieje online !!!
	//A258 - Pracovisko 2 - Ventilovy termnal VT2 nieje online !!!
    //A259 - Pracovisko 2 - Ventilovy termnal VT3 nieje online !!!
    //A260 - ST5_Srobovanie - Skrutkovacka M4 nieje online !!!
    //A261 - ST5_Srobovanie - Skrutkovacka M5 nieje online !!!
    //A262 - ST5_Srobovanie - Skrutkovacka M6 nieje online !!!
    //A263 - ST4_Maticovacka - Maticovacka M4 nieje online !!!
    //A264 - Pracovisko 2 - Kamery KAM1, KAM7, KAM10, KAM11, KAM12 a KAM17 niesu online !!!
    //A265 - Pracovisko 2 - Kamera KAM8 nieje online !!!
    //A266 - Pracovisko 2 - Kamera KAM9 nieje online !!!
    //A267 - ST4_Maticovacka - Porucha maticovacky M4 !!!
    //A268 - ST5_Srobovanie - Porucha vysunutia skrutkovacky M4 !!!
    //A269 - ST5_Srobovanie - Porucha vysunutia skrutkovacky M5 !!!
    //A270 - ST5_Srobovanie - Porucha vysunutia skrutkovacky M6 !!!
    //A271 - P2_Robot - porucha !!!
    //A272 - ST5_Srobovanie - Presiahnuty cas skrutkovania skrutky M4 !!!
    //A273 - ST5_Srobovanie - Presiahnuty cas skrutkovania skrutky M5 !!!
    //A274 - ST5_Srobovanie - Presiahnuty cas skrutkovania skrutky M6 !!!
    //A275 - ST5_Srobovanie - Skrutkovacka M4 nieje READY !!!
    //A276 - ST5_Srobovanie - Skrutkovacka M5 nieje READY !!!
    //A277 - ST5_Srobovanie - Skrutkovacka M6 nieje READY !!!
    //A278 - Pracovisko 2 - Prekrocena teplota motora vrchneho dopravnika !!!
    //A279 - Pracovisko 2 - Prekrocena teplota motora spodneho dopravnika !!!
    //A280 - Pracovisko 2 - Narusenie optickej bariery na vystupe !!!
    //A281 - Pracovisko 2 - Bolo stlacene tlacitko CS na ovladacom paneli !!!
    //A282 - Pracovisko 2 - Bolo stlacene tlacitko CS na rozvodnej skrini !!!
    //A283 - Pracovisko 2 - Bolo stlacene tlacitko CS robota !!!
    //A284 - Pracovisko 2 - Bolo stlacene tlacitko CS na dvojrucnom ovladani !!!
    //A285 - P2_Robot - Porucha odobratia Top Coveru z paletky !!!
    //A286 - ST3_Zakladanie tesnenia - Porucha vyvezenia paletky zo stopra !!!
    //A287 - ST4_Maticovacka - Porucha vyvezenia paletky zo stopra !!!
	//A288 - ST5_Srobovanie - Porucha vyvezenia paletky zo stopra !!!
    //A289 - ST6_Zvaranie - Porucha vyvezenia paletky zo stopra !!!
    //A290 - ST3_Zakladanie tesnenia - Porucha komunikacie s kamerou CAM 1 !!!
    //A291 - ST3_Zakladanie tesnenia - Porucha komunikacie s kamerou CAM 7 !!!
    //A292 - ST3_Zakladanie tesnenia - Porucha komunikacie s kamerou CAM 8 !!!
    //A293 - ST3_Zakladanie tesnenia - Porucha komunikacie s kamerou CAM 17 !!!
    //A294 - ST4_Maticovacka - Porucha komunikacie s kamerou CAM 9 !!!
    //A295 - ST5_Srobovanie - Porucha komunikacie s kamerou CAM 10 !!!
    //A296 - ST6_Zvaranie - Porucha komunikacie s kamerou CAM 11 !!!
    //A297 - ST6_Zvaranie - Porucha komunikacie s kamerou CAM 12 !!!

	//***************************Príznak pracovisko 2 stav PORUCHA**********************************//

    FOR a:=200 TO 299 BY 1 DO
        P2_Alarmy[a];
        IF P2_Alarmy[a] = TRUE THEN
            P2_Pracovisko.STAV.PORUCHA:= TRUE;
        END_IF
    END_FOR

    //*********************Pracovisko 2 - Porucha tlaku vzduchu*********************************//
    IF CasKontroly_TlakVzduchu.Q THEN
        P2_Alarmy[245]:= TRUE;
        P2_PoruchaST1:= TRUE;
        P2_PoruchaST2:= TRUE;
        P2_PoruchaST3:= TRUE;
        P2_PoruchaST4:= TRUE;
    END_IF

    IF Safety.STAV.P2_ZonaBunky_AKTIVNA AND NOT P2_Pracovisko.IN.PrivodVzduchu_SnimacTlaku_S3 THEN
        CasKontroly_TlakVzduchu.IN:= TRUE;
    ELSE
        CasKontroly_TlakVzduchu.IN:= FALSE;
    END_IF

    CasKontroly_TlakVzduchu.PT:= T#10s;
    CasKontroly_TlakVzduchu();

    //**********************************Porucha - kamerovy systém nieje online****************************************//
    IF CasKontroly_KAMsystem.Q THEN
        IF NOT Linka.STAV.WenglorControlUnit_OK THEN
            P2_Alarmy[264]:= TRUE;
            P2_PoruchaST1:= TRUE;
            P2_PoruchaST2:= TRUE;
            P2_PoruchaST3:= TRUE;
            P2_PoruchaST4:= TRUE;
        END_IF
        IF NOT CAM8.STAV.READY THEN
            P2_Alarmy[265]:= TRUE;
            P2_PoruchaST1:= TRUE;
        END_IF
        IF NOT CAM9.STAV.READY THEN
            P2_Alarmy[266]:= TRUE;
            P2_PoruchaST2:= TRUE;
        END_IF
    END_IF

    IF Safety.STAV.P2_ZonaBunky_AKTIVNA AND NOT P2_Pracovisko.STAV.Kamery_OK THEN
        CasKontroly_KAMsystem.IN:= TRUE;
    ELSE
        CasKontroly_KAMsystem.IN:= FALSE;
    END_IF

    CasKontroly_KAMsystem.PT:= T#2s;
    CasKontroly_KAMsystem();

    //**********************************Porucha - moduly niesu online**************************************************//
    IF CasKontroly_Moduly.Q THEN
        IF NOT P2_Pracovisko.STAV.ModulDI21_OK THEN
            P2_Alarmy[246]:= TRUE;
            P2_PoruchaST1:= TRUE;
            P2_PoruchaST2:= TRUE;
            P2_PoruchaST3:= TRUE;
            P2_PoruchaST4:= TRUE;
        END_IF
        IF NOT P2_Pracovisko.STAV.ModulDI22_OK THEN
            P2_Alarmy[247]:= TRUE;
            P2_PoruchaST1:= TRUE;
            P2_PoruchaST2:= TRUE;
            P2_PoruchaST3:= TRUE;
            P2_PoruchaST4:= TRUE;
        END_IF
        IF NOT P2_Pracovisko.STAV.ModulDI23_OK THEN
            P2_Alarmy[248]:= TRUE;
            P2_PoruchaST1:= TRUE;
            P2_PoruchaST2:= TRUE;
            P2_PoruchaST3:= TRUE;
            P2_PoruchaST4:= TRUE;
        END_IF
        IF NOT P2_Pracovisko.STAV.ModulDI24_OK THEN
            P2_Alarmy[249]:= TRUE;
            P2_PoruchaST1:= TRUE;
            P2_PoruchaST2:= TRUE;
            P2_PoruchaST3:= TRUE;
            P2_PoruchaST4:= TRUE;
        END_IF
        IF NOT P2_Pracovisko.STAV.ModulDI25_OK THEN
            P2_Alarmy[250]:= TRUE;
            P2_PoruchaST1:= TRUE;
            P2_PoruchaST2:= TRUE;
            P2_PoruchaST3:= TRUE;
            P2_PoruchaST4:= TRUE;
        END_IF
        IF NOT P2_Pracovisko.STAV.ModulDM21_OK THEN
            P2_Alarmy[251]:= TRUE;
            P2_PoruchaST1:= TRUE;
            P2_PoruchaST2:= TRUE;
            P2_PoruchaST3:= TRUE;
            P2_PoruchaST4:= TRUE;
        END_IF
        IF NOT P2_Pracovisko.STAV.ModulDS21_OK THEN
            P2_Alarmy[252]:= TRUE;
            P2_PoruchaST1:= TRUE;
            P2_PoruchaST2:= TRUE;
            P2_PoruchaST3:= TRUE;
            P2_PoruchaST4:= TRUE;
        END_IF
        IF NOT P2_Pracovisko.STAV.ModulDS22_OK THEN
            P2_Alarmy[253]:= TRUE;
            P2_PoruchaST1:= TRUE;
            P2_PoruchaST2:= TRUE;
            P2_PoruchaST3:= TRUE;
            P2_PoruchaST4:= TRUE;
        END_IF
        IF NOT P2_Pracovisko.STAV.ModulDS23_OK THEN
            P2_Alarmy[254]:= TRUE;
            P2_PoruchaST1:= TRUE;
            P2_PoruchaST2:= TRUE;
            P2_PoruchaST3:= TRUE;
            P2_PoruchaST4:= TRUE;
        END_IF
        IF NOT P2_Pracovisko.STAV.ModulSI21_OK THEN
            P2_Alarmy[255]:= TRUE;
            P2_PoruchaST1:= TRUE;
            P2_PoruchaST2:= TRUE;
            P2_PoruchaST3:= TRUE;
            P2_PoruchaST4:= TRUE;
        END_IF
        IF NOT P2_Pracovisko.STAV.ModulSI22_OK THEN
            P2_Alarmy[256]:= TRUE;
            P2_PoruchaST1:= TRUE;
            P2_PoruchaST2:= TRUE;
            P2_PoruchaST3:= TRUE;
            P2_PoruchaST4:= TRUE;
        END_IF
    END_IF

    IF Safety.STAV.P2_ZonaBunky_AKTIVNA AND NOT P2_Pracovisko.STAV.Moduly_OK THEN
        CasKontroly_Moduly.IN:= TRUE;
    ELSE
        CasKontroly_Moduly.IN:= FALSE;
    END_IF

    CasKontroly_Moduly.PT:= T#2s;
    CasKontroly_Moduly();

    //********************************Porucha - ventilové terminály niesu online**********************************************//
    IF CasKontroly_VentTerminalov.Q THEN
        IF NOT P2_Pracovisko.STAV.VentilovyTerminal_VT1_OK THEN
            P2_Alarmy[257]:= TRUE;
            P2_PoruchaST1:= TRUE;
            P2_PoruchaST2:= TRUE;
            P2_PoruchaST3:= TRUE;
            P2_PoruchaST4:= TRUE;
        END_IF
        IF NOT P2_Pracovisko.STAV.VentilovyTerminal_VT2_OK THEN
            P2_Alarmy[258]:= TRUE;
            P2_PoruchaST1:= TRUE;
            P2_PoruchaST2:= TRUE;
            P2_PoruchaST3:= TRUE;
            P2_PoruchaST4:= TRUE;
        END_IF
        IF NOT P2_Pracovisko.STAV.VentilovyTerminal_VT3_OK THEN
            P2_Alarmy[259]:= TRUE;
            P2_PoruchaST1:= TRUE;
            P2_PoruchaST2:= TRUE;
            P2_PoruchaST3:= TRUE;
            P2_PoruchaST4:= TRUE;
        END_IF
    END_IF

    IF Safety.STAV.P2_ZonaBunky_AKTIVNA AND NOT P2_Pracovisko.STAV.VentiloveTerminaly_OK THEN
        CasKontroly_VentTerminalov.IN:= TRUE;
    ELSE
        CasKontroly_VentTerminalov.IN:= FALSE;
    END_IF

    CasKontroly_VentTerminalov.PT:= T#2s;
    CasKontroly_VentTerminalov();

    //********************************Porucha - skrutkovacky niesu online**********************************************//
    IF CasKontroly_Skrutkovacky.Q THEN
        IF NOT P2_Pracovisko.STAV.Skrutkovacka_M4_OK THEN
            P2_Alarmy[260]:= TRUE;
            P2_PoruchaST3:= TRUE;
        END_IF
        IF NOT P2_Pracovisko.STAV.Skrutkovacka_M5_OK THEN
            P2_Alarmy[261]:= TRUE;
            P2_PoruchaST3:= TRUE;
        END_IF
        IF NOT P2_Pracovisko.STAV.Skrutkovacka_M6_OK THEN
            P2_Alarmy[262]:= TRUE;
            P2_PoruchaST3:= TRUE;
        END_IF
        IF NOT P2_Pracovisko.STAV.Maticovacka_M4_OK THEN
            P2_Alarmy[263]:= TRUE;
            P2_PoruchaST2:= TRUE;
        END_IF
    END_IF

    IF Safety.STAV.P2_ZonaBunky_AKTIVNA AND NOT P2_Pracovisko.STAV.Skrutkovacky_OK THEN
        CasKontroly_Skrutkovacky.IN:= TRUE;
    ELSE
        CasKontroly_Skrutkovacky.IN:= FALSE;
    END_IF

    CasKontroly_Skrutkovacky.PT:= T#2s;
    CasKontroly_Skrutkovacky();

    //*********************************Porucha - robot nieje online************************************************//
    IF CasKontroly_Robota.Q THEN
        P2_Alarmy[244]:= TRUE;
        P2_PoruchaST3:= TRUE;
        P2_PoruchaST4:= TRUE;
    END_IF

    IF Safety.STAV.P2_ZonaBunky_AKTIVNA AND NOT P2_Pracovisko.STAV.KOM_Robot_OK THEN
        CasKontroly_Robota.IN:= TRUE;
    ELSE
        CasKontroly_Robota.IN:= FALSE;
    END_IF

    CasKontroly_Robota.PT:= T#2s;
    CasKontroly_Robota();

    //*******************************Porucha napájania robota*****************************************************//
    IF CasKontroly_Robota.Q AND NOT P2_Pracovisko.IN.NapajaniaRobota_OK THEN
        P2_Alarmy[243]:= TRUE;
        P2_PoruchaST3:= TRUE;
        P2_PoruchaST4:= TRUE;
    END_IF

    //********************Pracovisko 2 - Porucha ochrannej bariéry zdvihu zakladača tesnenia****************************************//
    IF Safety.IN.P2_ZaklTesnenia_Zdvih_BUSY AND NOT Safety.STAV.P2_ZaklTesnenia_Bariera_AKTIVNA THEN
        P2_Alarmy[206]:= TRUE;
        P2_PoruchaST1:= TRUE;
    END_IF

    //*********************Pracovisko 2 - Porucha serva zdvihu zakladača tesnenia***************//
    IF CasPoruchyServaZdvihuZakladaca.Q THEN
        P2_Alarmy[202]:= TRUE;
        P2_PoruchaST1:= TRUE;
	END_IF

    IF Safety.STAV.P2_ZonaZaklTesnenZdvih_AKTIVNA AND P2_ZakladacTesnenia.ServoZdvihuZakladaca_M4.STATUS.ERROR THEN
        CasPoruchyServaZdvihuZakladaca.IN:= TRUE;
    ELSE
        CasPoruchyServaZdvihuZakladaca.IN:= FALSE;
    END_IF

    CasPoruchyServaZdvihuZakladaca.PT:= T#2s;
    CasPoruchyServaZdvihuZakladaca();

    //********************Pracovisko 2 - Porucha bumpera suflíka zakladača tesnenia****************************************//
    IF Safety.IN.P2_ZaklTesnenia_Vysuvanie_BUSY AND NOT Safety.STAV.P2_ZaklTesnenia_Bumper_AKTIVNY THEN
        P2_Alarmy[207]:= TRUE;
        P2_PoruchaST1:= TRUE;
    END_IF

	//*********************Pracovisko 2 - Porucha serva pojazdu zakladača tesnenia***************//
	IF CasPoruchyServaPojazduZakladaca.Q THEN
        P2_Alarmy[203]:= TRUE;
        P2_PoruchaST1:= TRUE;
	END_IF

    IF Safety.STAV.P2_ZonaZaklTesnenPojazd_AKTIVNA AND P2_ZakladacTesnenia.ServoPojazduVozika_M5.STATUS.ERROR THEN
        CasPoruchyServaPojazduZakladaca.IN:= TRUE;
    ELSE
        CasPoruchyServaPojazduZakladaca.IN:= FALSE;
    END_IF

    CasPoruchyServaPojazduZakladaca.PT:= T#2s;
    CasPoruchyServaPojazduZakladaca();

	//*********************Pracovisko 2 - Porucha serva manipulatora šrobovania os X***************//
	IF CasPoruchyServaSrobovaniaOsX.Q THEN
        P2_Alarmy[215]:= TRUE;
        P2_PoruchaST3:= TRUE;
	END_IF

    IF Safety.STAV.P2_ZonaBunky_AKTIVNA AND P2_Srobovanie.ServoManipulOsX_M10.STATUS.ERROR THEN
        CasPoruchyServaSrobovaniaOsX.IN:= TRUE;
    ELSE
        CasPoruchyServaSrobovaniaOsX.IN:= FALSE;
    END_IF

    CasPoruchyServaSrobovaniaOsX.PT:= T#2s;
    CasPoruchyServaSrobovaniaOsX();

	//*********************Pracovisko 2 - Porucha serva manipulatora šrobovania os Y***************//
	IF CasPoruchyServaSrobovaniaOsY.Q THEN
        P2_Alarmy[216]:= TRUE;
        P2_PoruchaST3:= TRUE;
	END_IF

    IF Safety.STAV.P2_ZonaBunky_AKTIVNA AND P2_Srobovanie.ServoManipulOsY_M9.STATUS.ERROR THEN
        CasPoruchyServaSrobovaniaOsY.IN:= TRUE;
    ELSE
        CasPoruchyServaSrobovaniaOsY.IN:= FALSE;
    END_IF

    CasPoruchyServaSrobovaniaOsY.PT:= T#2s;
    CasPoruchyServaSrobovaniaOsY();

	//**********************Pracovisko 2 - Porucha serva zdvihu zvarania****************************//
	IF CasPoruchyServaZdvihuZvarania.Q THEN
        P2_Alarmy[220]:= TRUE;
        P2_PoruchaST4:= TRUE;
	END_IF

    IF Safety.STAV.P2_ZonaBunky_AKTIVNA AND P2_Zvaranie.ServoZdvihuZvarania_M6.STATUS.ERROR THEN
        CasPoruchyServaZdvihuZvarania.IN:= TRUE;
    ELSE
        CasPoruchyServaZdvihuZvarania.IN:= FALSE;
    END_IF

    CasPoruchyServaZdvihuZvarania.PT:= T#2s;
    CasPoruchyServaZdvihuZvarania();

    //****************************Pracovisko 2 - porucha vrchného dopravníka**********************************//
    IF NOT P2_Dopravniky.IN.HornyDoprav_TeplotaMotora_OK AND P2_Pracovisko.STAV.Automat THEN
        P2_Alarmy[278]:= TRUE;
    END_IF

    //*****************************Pracovisko 2 - porucha spodného dopravníka************************************//
    IF NOT P2_Dopravniky.IN.SpodnyDoprav_TeplotaMotora_OK AND P2_Pracovisko.STAV.Automat THEN
        P2_Alarmy[279]:= TRUE;
    END_IF

    //******************************Pracovisko 2 - narušenie výstupnej bariery***********************************//
    IF NOT Safety.STAV.P3_VstupBunky_Bariera_AKTIVNA AND NOT Safety.STAV.P3_ZonaBunky_AKTIVNA AND P2_Pracovisko.STAV.Automat THEN
        P2_Alarmy[280]:= TRUE;
    END_IF

    //******************************Stlačenie tlačítok CS*******************************************************//
    IF EDGENEG(Safety.STAV.P2_Panel_TlacitkoCS_AKTIVNE) THEN
        P2_Alarmy[281]:= TRUE;
    END_IF

    IF EDGENEG(Safety.STAV.P2_Skrina_TlacitkoCS_AKTIVNE) THEN
        P2_Alarmy[282]:= TRUE;
    END_IF

    IF EDGENEG(Safety.STAV.P2_Robot_TlacitkoCS_AKTIVNE) THEN
        P2_Alarmy[283]:= TRUE;
    END_IF

    IF EDGENEG(Safety.STAV.P2_TlacitkoCS_AKTIVNE) THEN
        P2_Alarmy[284]:= TRUE;
    END_IF

    //***************************************************Nasetovanie alarmov****************************************************//

	IF P2_Alarmy[200] THEN
		MpAlarmXSet(gAlarmXCore, 'A200');
	ELSE
		MpAlarmXReset(gAlarmXCore, 'A200');
	END_IF

	IF P2_Alarmy[201] THEN
		MpAlarmXSet(gAlarmXCore, 'A201');
	ELSE
		MpAlarmXReset(gAlarmXCore, 'A201');
	END_IF

	IF P2_Alarmy[202] THEN
		MpAlarmXSet(gAlarmXCore, 'A202');
	ELSE
		MpAlarmXReset(gAlarmXCore, 'A202');
	END_IF

	IF P2_Alarmy[203] THEN
		MpAlarmXSet(gAlarmXCore, 'A203');
	ELSE
		MpAlarmXReset(gAlarmXCore, 'A203');
	END_IF

	IF P2_Alarmy[204] THEN
		MpAlarmXSet(gAlarmXCore, 'A204');
	ELSE
		MpAlarmXReset(gAlarmXCore, 'A204');
	END_IF

	IF P2_Alarmy[205] THEN
		MpAlarmXSet(gAlarmXCore, 'A205');
	ELSE
		MpAlarmXReset(gAlarmXCore, 'A205');
	END_IF

	IF P2_Alarmy[206] THEN
		MpAlarmXSet(gAlarmXCore, 'A206');
	ELSE
		MpAlarmXReset(gAlarmXCore, 'A206');
	END_IF

	IF P2_Alarmy[207] THEN
		MpAlarmXSet(gAlarmXCore, 'A207');
	ELSE
		MpAlarmXReset(gAlarmXCore, 'A207');
	END_IF

	IF P2_Alarmy[208] THEN
		MpAlarmXSet(gAlarmXCore, 'A208');
	ELSE
		MpAlarmXReset(gAlarmXCore, 'A208');
	END_IF

	IF P2_Alarmy[209] THEN
		MpAlarmXSet(gAlarmXCore, 'A209');
	ELSE
		MpAlarmXReset(gAlarmXCore, 'A209');
	END_IF

	IF P2_Alarmy[210] THEN
		MpAlarmXSet(gAlarmXCore, 'A210');
	ELSE
		MpAlarmXReset(gAlarmXCore, 'A210');
	END_IF

	IF P2_Alarmy[211] THEN
		MpAlarmXSet(gAlarmXCore, 'A211');
	ELSE
		MpAlarmXReset(gAlarmXCore, 'A211');
	END_IF

	IF P2_Alarmy[212] THEN
		MpAlarmXSet(gAlarmXCore, 'A212');
	ELSE
		MpAlarmXReset(gAlarmXCore, 'A212');
	END_IF

	IF P2_Alarmy[213] THEN
		MpAlarmXSet(gAlarmXCore, 'A213');
	ELSE
		MpAlarmXReset(gAlarmXCore, 'A213');
	END_IF

	IF P2_Alarmy[214] THEN
		MpAlarmXSet(gAlarmXCore, 'A214');
	ELSE
		MpAlarmXReset(gAlarmXCore, 'A214');
	END_IF

	IF P2_Alarmy[215] THEN
		MpAlarmXSet(gAlarmXCore, 'A215');
	ELSE
		MpAlarmXReset(gAlarmXCore, 'A215');
	END_IF

	IF P2_Alarmy[216] THEN
		MpAlarmXSet(gAlarmXCore, 'A216');
	ELSE
		MpAlarmXReset(gAlarmXCore, 'A216');
	END_IF

	IF P2_Alarmy[217] THEN
		MpAlarmXSet(gAlarmXCore, 'A217');
	ELSE
		MpAlarmXReset(gAlarmXCore, 'A217');
	END_IF

	IF P2_Alarmy[218] THEN
		MpAlarmXSet(gAlarmXCore, 'A218');
	ELSE
		MpAlarmXReset(gAlarmXCore, 'A218');
	END_IF

	IF P2_Alarmy[219] THEN
		MpAlarmXSet(gAlarmXCore, 'A219');
	ELSE
		MpAlarmXReset(gAlarmXCore, 'A219');
	END_IF

	IF P2_Alarmy[220] THEN
		MpAlarmXSet(gAlarmXCore, 'A220');
	ELSE
		MpAlarmXReset(gAlarmXCore, 'A220');
	END_IF

	IF P2_Alarmy[221] THEN
		MpAlarmXSet(gAlarmXCore, 'A221');
	ELSE
		MpAlarmXReset(gAlarmXCore, 'A221');
	END_IF

	IF P2_Alarmy[222] THEN
		MpAlarmXSet(gAlarmXCore, 'A222');
	ELSE
		MpAlarmXReset(gAlarmXCore, 'A222');
	END_IF

	IF P2_Alarmy[223] THEN
		MpAlarmXSet(gAlarmXCore, 'A223');
	ELSE
		MpAlarmXReset(gAlarmXCore, 'A223');
	END_IF

	IF P2_Alarmy[224] THEN
		MpAlarmXSet(gAlarmXCore, 'A224');
	ELSE
		MpAlarmXReset(gAlarmXCore, 'A224');
	END_IF

	IF P2_Alarmy[225] THEN
		MpAlarmXSet(gAlarmXCore, 'A225');
	ELSE
		MpAlarmXReset(gAlarmXCore, 'A225');
	END_IF

	IF P2_Alarmy[226] THEN
		MpAlarmXSet(gAlarmXCore, 'A226');
	ELSE
		MpAlarmXReset(gAlarmXCore, 'A226');
	END_IF

	IF P2_Alarmy[227] THEN
		MpAlarmXSet(gAlarmXCore, 'A227');
	ELSE
		MpAlarmXReset(gAlarmXCore, 'A227');
	END_IF

	IF P2_Alarmy[228] THEN
		MpAlarmXSet(gAlarmXCore, 'A228');
	ELSE
		MpAlarmXReset(gAlarmXCore, 'A228');
	END_IF

	IF P2_Alarmy[229] THEN
		MpAlarmXSet(gAlarmXCore, 'A229');
	ELSE
		MpAlarmXReset(gAlarmXCore, 'A229');
	END_IF

	IF P2_Alarmy[230] THEN
		MpAlarmXSet(gAlarmXCore, 'A230');
	ELSE
		MpAlarmXReset(gAlarmXCore, 'A230');
	END_IF

    IF P2_Alarmy[231] THEN
        MpAlarmXSet(gAlarmXCore, 'A231');
    ELSE
        MpAlarmXReset(gAlarmXCore, 'A231');
    END_IF

    IF P2_Alarmy[232] THEN
        MpAlarmXSet(gAlarmXCore, 'A232');
    ELSE
        MpAlarmXReset(gAlarmXCore, 'A232');
    END_IF

    IF P2_Alarmy[233] THEN
        MpAlarmXSet(gAlarmXCore, 'A233');
    ELSE
        MpAlarmXReset(gAlarmXCore, 'A233');
    END_IF

    IF P2_Alarmy[234] THEN
        MpAlarmXSet(gAlarmXCore, 'A234');
    ELSE
        MpAlarmXReset(gAlarmXCore, 'A234');
    END_IF

    IF P2_Alarmy[235] THEN
        MpAlarmXSet(gAlarmXCore, 'A235');
    ELSE
        MpAlarmXReset(gAlarmXCore, 'A235');
    END_IF

    IF P2_Alarmy[236] THEN
        MpAlarmXSet(gAlarmXCore, 'A236');
    ELSE
        MpAlarmXReset(gAlarmXCore, 'A236');
    END_IF

    IF P2_Alarmy[237] THEN
        MpAlarmXSet(gAlarmXCore, 'A237');
    ELSE
        MpAlarmXReset(gAlarmXCore, 'A237');
    END_IF

    IF P2_Alarmy[238] THEN
        MpAlarmXSet(gAlarmXCore, 'A238');
    ELSE
        MpAlarmXReset(gAlarmXCore, 'A238');
    END_IF

    IF P2_Alarmy[239] THEN
        MpAlarmXSet(gAlarmXCore, 'A239');
    ELSE
        MpAlarmXReset(gAlarmXCore, 'A239');
    END_IF

    IF P2_Alarmy[240] THEN
        MpAlarmXSet(gAlarmXCore, 'A240');
    ELSE
        MpAlarmXReset(gAlarmXCore, 'A240');
    END_IF

    IF P2_Alarmy[241] THEN
        MpAlarmXSet(gAlarmXCore, 'A241');
    ELSE
        MpAlarmXReset(gAlarmXCore, 'A241');
    END_IF

    IF P2_Alarmy[242] THEN
        MpAlarmXSet(gAlarmXCore, 'A242');
    ELSE
        MpAlarmXReset(gAlarmXCore, 'A242');
    END_IF

    IF P2_Alarmy[243] THEN
        MpAlarmXSet(gAlarmXCore, 'A243');
    ELSE
        MpAlarmXReset(gAlarmXCore, 'A243');
    END_IF

    IF P2_Alarmy[244] THEN
        MpAlarmXSet(gAlarmXCore, 'A244');
    ELSE
        MpAlarmXReset(gAlarmXCore, 'A244');
    END_IF

    IF P2_Alarmy[245] THEN
        MpAlarmXSet(gAlarmXCore, 'A245');
    ELSE
        MpAlarmXReset(gAlarmXCore, 'A245');
    END_IF

    IF P2_Alarmy[246] THEN
        MpAlarmXSet(gAlarmXCore, 'A246');
    ELSE
        MpAlarmXReset(gAlarmXCore, 'A246');
    END_IF

    IF P2_Alarmy[247] THEN
        MpAlarmXSet(gAlarmXCore, 'A247');
    ELSE
        MpAlarmXReset(gAlarmXCore, 'A247');
    END_IF

    IF P2_Alarmy[248] THEN
        MpAlarmXSet(gAlarmXCore, 'A248');
    ELSE
        MpAlarmXReset(gAlarmXCore, 'A248');
    END_IF

    IF P2_Alarmy[249] THEN
        MpAlarmXSet(gAlarmXCore, 'A249');
    ELSE
        MpAlarmXReset(gAlarmXCore, 'A249');
    END_IF

    IF P2_Alarmy[250] THEN
        MpAlarmXSet(gAlarmXCore, 'A250');
    ELSE
        MpAlarmXReset(gAlarmXCore, 'A250');
    END_IF

    IF P2_Alarmy[251] THEN
        MpAlarmXSet(gAlarmXCore, 'A251');
    ELSE
        MpAlarmXReset(gAlarmXCore, 'A251');
    END_IF

    IF P2_Alarmy[252] THEN
        MpAlarmXSet(gAlarmXCore, 'A252');
    ELSE
        MpAlarmXReset(gAlarmXCore, 'A252');
    END_IF

    IF P2_Alarmy[253] THEN
        MpAlarmXSet(gAlarmXCore, 'A253');
    ELSE
        MpAlarmXReset(gAlarmXCore, 'A253');
    END_IF

    IF P2_Alarmy[254] THEN
        MpAlarmXSet(gAlarmXCore, 'A254');
    ELSE
        MpAlarmXReset(gAlarmXCore, 'A254');
    END_IF

    IF P2_Alarmy[255] THEN
        MpAlarmXSet(gAlarmXCore, 'A255');
    ELSE
        MpAlarmXReset(gAlarmXCore, 'A255');
    END_IF

    IF P2_Alarmy[256] THEN
        MpAlarmXSet(gAlarmXCore, 'A256');
    ELSE
        MpAlarmXReset(gAlarmXCore, 'A256');
    END_IF

    IF P2_Alarmy[257] THEN
        MpAlarmXSet(gAlarmXCore, 'A257');
    ELSE
        MpAlarmXReset(gAlarmXCore, 'A257');
    END_IF

    IF P2_Alarmy[258] THEN
        MpAlarmXSet(gAlarmXCore, 'A258');
    ELSE
        MpAlarmXReset(gAlarmXCore, 'A258');
    END_IF

    IF P2_Alarmy[259] THEN
        MpAlarmXSet(gAlarmXCore, 'A259');
    ELSE
        MpAlarmXReset(gAlarmXCore, 'A259');
    END_IF

    IF P2_Alarmy[260] THEN
        MpAlarmXSet(gAlarmXCore, 'A260');
    ELSE
        MpAlarmXReset(gAlarmXCore, 'A260');
    END_IF

    IF P2_Alarmy[261] THEN
        MpAlarmXSet(gAlarmXCore, 'A261');
    ELSE
        MpAlarmXReset(gAlarmXCore, 'A261');
    END_IF

    IF P2_Alarmy[262] THEN
        MpAlarmXSet(gAlarmXCore, 'A262');
    ELSE
        MpAlarmXReset(gAlarmXCore, 'A262');
    END_IF

    IF P2_Alarmy[263] THEN
        MpAlarmXSet(gAlarmXCore, 'A263');
    ELSE
        MpAlarmXReset(gAlarmXCore, 'A263');
    END_IF

    IF P2_Alarmy[264] THEN
        MpAlarmXSet(gAlarmXCore, 'A264');
    ELSE
        MpAlarmXReset(gAlarmXCore, 'A264');
    END_IF

    IF P2_Alarmy[265] THEN
        MpAlarmXSet(gAlarmXCore, 'A265');
    ELSE
        MpAlarmXReset(gAlarmXCore, 'A265');
    END_IF

    IF P2_Alarmy[266] THEN
        MpAlarmXSet(gAlarmXCore, 'A266');
    ELSE
        MpAlarmXReset(gAlarmXCore, 'A266');
    END_IF

    IF P2_Alarmy[267] THEN
        MpAlarmXSet(gAlarmXCore, 'A267');
    ELSE
        MpAlarmXReset(gAlarmXCore, 'A267');
    END_IF

    IF P2_Alarmy[268] THEN
        MpAlarmXSet(gAlarmXCore, 'A268');
    ELSE
        MpAlarmXReset(gAlarmXCore, 'A268');
    END_IF

    IF P2_Alarmy[269] THEN
        MpAlarmXSet(gAlarmXCore, 'A269');
    ELSE
        MpAlarmXReset(gAlarmXCore, 'A269');
    END_IF

    IF P2_Alarmy[270] THEN
        MpAlarmXSet(gAlarmXCore, 'A270');
    ELSE
        MpAlarmXReset(gAlarmXCore, 'A270');
    END_IF

    IF P2_Alarmy[271] THEN
        MpAlarmXSet(gAlarmXCore, 'A271');
    ELSE
        MpAlarmXReset(gAlarmXCore, 'A271');
    END_IF

    IF P2_Alarmy[272] THEN
        MpAlarmXSet(gAlarmXCore, 'A272');
    ELSE
        MpAlarmXReset(gAlarmXCore, 'A272');
    END_IF

    IF P2_Alarmy[273] THEN
        MpAlarmXSet(gAlarmXCore, 'A273');
    ELSE
        MpAlarmXReset(gAlarmXCore, 'A273');
    END_IF

    IF P2_Alarmy[274] THEN
        MpAlarmXSet(gAlarmXCore, 'A274');
    ELSE
        MpAlarmXReset(gAlarmXCore, 'A274');
    END_IF

    IF P2_Alarmy[275] THEN
        MpAlarmXSet(gAlarmXCore, 'A275');
    ELSE
        MpAlarmXReset(gAlarmXCore, 'A275');
    END_IF

    IF P2_Alarmy[276] THEN
        MpAlarmXSet(gAlarmXCore, 'A276');
    ELSE
        MpAlarmXReset(gAlarmXCore, 'A276');
    END_IF

    IF P2_Alarmy[277] THEN
        MpAlarmXSet(gAlarmXCore, 'A277');
    ELSE
        MpAlarmXReset(gAlarmXCore, 'A277');
    END_IF

    IF P2_Alarmy[278] THEN
        MpAlarmXSet(gAlarmXCore, 'A278');
    ELSE
        MpAlarmXReset(gAlarmXCore, 'A278');
    END_IF

    IF P2_Alarmy[279] THEN
        MpAlarmXSet(gAlarmXCore, 'A279');
    ELSE
        MpAlarmXReset(gAlarmXCore, 'A279');
    END_IF

    IF P2_Alarmy[280] THEN
        MpAlarmXSet(gAlarmXCore, 'A280');
    ELSE
        MpAlarmXReset(gAlarmXCore, 'A280');
    END_IF

    IF P2_Alarmy[281] THEN
        MpAlarmXSet(gAlarmXCore, 'A281');
    ELSE
        MpAlarmXReset(gAlarmXCore, 'A281');
    END_IF

    IF P2_Alarmy[282] THEN
        MpAlarmXSet(gAlarmXCore, 'A282');
    ELSE
        MpAlarmXReset(gAlarmXCore, 'A282');
    END_IF

    IF P2_Alarmy[283] THEN
        MpAlarmXSet(gAlarmXCore, 'A283');
    ELSE
        MpAlarmXReset(gAlarmXCore, 'A283');
    END_IF

    IF P2_Alarmy[284] THEN
        MpAlarmXSet(gAlarmXCore, 'A284');
    ELSE
        MpAlarmXReset(gAlarmXCore, 'A284');
    END_IF

    IF P2_Alarmy[285] THEN
        MpAlarmXSet(gAlarmXCore, 'A285');
    ELSE
        MpAlarmXReset(gAlarmXCore, 'A285');
    END_IF

    IF P2_Alarmy[286] THEN
        MpAlarmXSet(gAlarmXCore, 'A286');
    ELSE
        MpAlarmXReset(gAlarmXCore, 'A286');
    END_IF

    IF P2_Alarmy[287] THEN
        MpAlarmXSet(gAlarmXCore, 'A287');
    ELSE
        MpAlarmXReset(gAlarmXCore, 'A287');
    END_IF

    IF P2_Alarmy[288] THEN
        MpAlarmXSet(gAlarmXCore, 'A288');
    ELSE
        MpAlarmXReset(gAlarmXCore, 'A288');
    END_IF

    IF P2_Alarmy[289] THEN
        MpAlarmXSet(gAlarmXCore, 'A289');
    ELSE
        MpAlarmXReset(gAlarmXCore, 'A289');
    END_IF

    IF P2_Alarmy[290] THEN
        MpAlarmXSet(gAlarmXCore, 'A290');
    ELSE
        MpAlarmXReset(gAlarmXCore, 'A290');
    END_IF

    IF P2_Alarmy[291] THEN
        MpAlarmXSet(gAlarmXCore, 'A291');
    ELSE
        MpAlarmXReset(gAlarmXCore, 'A291');
    END_IF

    IF P2_Alarmy[292] THEN
        MpAlarmXSet(gAlarmXCore, 'A292');
    ELSE
        MpAlarmXReset(gAlarmXCore, 'A292');
    END_IF

    IF P2_Alarmy[293] THEN
        MpAlarmXSet(gAlarmXCore, 'A293');
    ELSE
        MpAlarmXReset(gAlarmXCore, 'A293');
    END_IF

    IF P2_Alarmy[294] THEN
        MpAlarmXSet(gAlarmXCore, 'A294');
    ELSE
        MpAlarmXReset(gAlarmXCore, 'A294');
    END_IF

    IF P2_Alarmy[295] THEN
        MpAlarmXSet(gAlarmXCore, 'A295');
    ELSE
        MpAlarmXReset(gAlarmXCore, 'A295');
    END_IF

    IF P2_Alarmy[296] THEN
        MpAlarmXSet(gAlarmXCore, 'A296');
    ELSE
        MpAlarmXReset(gAlarmXCore, 'A296');
    END_IF

    IF P2_Alarmy[297] THEN
        MpAlarmXSet(gAlarmXCore, 'A297');
    ELSE
        MpAlarmXReset(gAlarmXCore, 'A297');
    END_IF

    //********************************Zobrazenie symbolu alarmu*****************************************************//

    IF P2_Pracovisko.STAV.PORUCHA THEN
        P2_AlarmyVizu.ZobrazSymbolAlarmu:= Blikac1s;
    ELSE
        P2_AlarmyVizu.ZobrazSymbolAlarmu:= FALSE;
    END_IF

    //********************************Blikanie tlačítka Alarmy*******************************************************//
    IF P2_Pracovisko.STAV.PORUCHA AND P2_Vizu.ActualPage <> 'PageAlarmP2' THEN
        IF Blikac1s THEN
            P2_AlarmyVizu.FarbaTlacitka_Alarmy:= "Button_Red";
        ELSE
            P2_AlarmyVizu.FarbaTlacitka_Alarmy:= "default";
        END_IF
    ELSE
        P2_AlarmyVizu.FarbaTlacitka_Alarmy:= "default";
    END_IF

	//*************************************Potvrdenie alarmov*********************************************************//
	IF P2_AlarmyVizu.PotvrdAlarmy THEN
		brsmemset(ADR(P2_Alarmy),0,SIZEOF(P2_Alarmy));
		P2_Pracovisko.STAV.PORUCHA:= FALSE;
		P2_PoruchaST1:= FALSE;
		P2_PoruchaST2:= FALSE;
		P2_PoruchaST3:= FALSE;
		P2_PoruchaST4:= FALSE;
		IF P2_ZakladacTesnenia.ServoZdvihuZakladaca_M4.STATUS.ERROR AND P2_ZakladacTesnenia.ServoZdvihuZakladaca_M4.STATUS.ReadyToPower_ON THEN
            P2_ZakladacTesnenia.ServoZdvihuZakladaca_M4.CMD.ErrorRESET:= TRUE;
        END_IF
        IF P2_ZakladacTesnenia.ServoPojazduVozika_M5.STATUS.ERROR AND P2_ZakladacTesnenia.ServoPojazduVozika_M5.STATUS.ReadyToPower_ON THEN
            P2_ZakladacTesnenia.ServoPojazduVozika_M5.CMD.ErrorRESET:= TRUE;
        END_IF
        IF P2_Srobovanie.ServoManipulOsX_M10.STATUS.ERROR AND P2_Srobovanie.ServoManipulOsX_M10.STATUS.ReadyToPower_ON THEN
            P2_Srobovanie.ServoManipulOsX_M10.CMD.ErrorRESET:= TRUE;
        END_IF
        IF P2_Srobovanie.ServoManipulOsY_M9.STATUS.ERROR AND P2_Srobovanie.ServoManipulOsY_M9.STATUS.ReadyToPower_ON THEN
            P2_Srobovanie.ServoManipulOsY_M9.CMD.ErrorRESET:= TRUE;
        END_IF
        IF P2_Zvaranie.ServoZdvihuZvarania_M6.STATUS.ERROR AND P2_Zvaranie.ServoZdvihuZvarania_M6.STATUS.ReadyToPower_ON THEN
            P2_Zvaranie.ServoZdvihuZvarania_M6.CMD.ErrorRESET:= TRUE;
        END_IF
		P2_AlarmyVizu.PotvrdAlarmy:= FALSE;
	END_IF

    //Resetovanie serv zakladača tesnenia//
    IF EDGEPOS(Safety.STAV.P2_ZonaZaklTesnenZdvih_AKTIVNA) THEN
        P2_ZakladacTesnenia.ServoZdvihuZakladaca_M4.CMD.ErrorRESET:= TRUE;
    END_IF

    IF EDGEPOS(Safety.STAV.P2_ZonaZaklTesnenPojazd_AKTIVNA) THEN
        P2_ZakladacTesnenia.ServoPojazduVozika_M5.CMD.ErrorRESET:= TRUE;
    END_IF

    //Resetovanie poruch serv pri zatvorení bunky//
    IF EDGEPOS(Safety.STAV.P2_ZonaBunky_AKTIVNA) THEN
        P2_Srobovanie.ServoManipulOsX_M10.CMD.ErrorRESET:= TRUE;
        P2_Srobovanie.ServoManipulOsY_M9.CMD.ErrorRESET:= TRUE;
        P2_Zvaranie.ServoZdvihuZvarania_M6.CMD.ErrorRESET:= TRUE;
    END_IF

    //Zrušenie resetovania porúch serv//
    IF NOT P2_ZakladacTesnenia.ServoZdvihuZakladaca_M4.STATUS.ERROR THEN
        P2_ZakladacTesnenia.ServoZdvihuZakladaca_M4.CMD.ErrorRESET:= FALSE;
    ELSIF CasResetServaZdvihuZakladaca.Q THEN
        P2_ZakladacTesnenia.ServoZdvihuZakladaca_M4.CMD.ErrorRESET:= FALSE;
    END_IF

    IF NOT P2_ZakladacTesnenia.ServoPojazduVozika_M5.STATUS.ERROR THEN
        P2_ZakladacTesnenia.ServoPojazduVozika_M5.CMD.ErrorRESET:= FALSE;
    ELSIF CasResetServaPojazduZakladaca.Q THEN
        P2_ZakladacTesnenia.ServoPojazduVozika_M5.CMD.ErrorRESET:= FALSE;
    END_IF

    IF NOT P2_Srobovanie.ServoManipulOsX_M10.STATUS.ERROR THEN
        P2_Srobovanie.ServoManipulOsX_M10.CMD.ErrorRESET:= FALSE;
    ELSIF CasResetovaniaServaSrobovaniaOsX.Q THEN
        P2_Srobovanie.ServoManipulOsX_M10.CMD.ErrorRESET:= FALSE;
    END_IF

    IF NOT P2_Srobovanie.ServoManipulOsY_M9.STATUS.ERROR THEN
        P2_Srobovanie.ServoManipulOsY_M9.CMD.ErrorRESET:= FALSE;
    ELSIF CasResetovaniaServaSrobovaniaOsY.Q THEN
        P2_Srobovanie.ServoManipulOsY_M9.CMD.ErrorRESET:= FALSE;
    END_IF

    IF NOT P2_Zvaranie.ServoZdvihuZvarania_M6.STATUS.ERROR THEN
        P2_Zvaranie.ServoZdvihuZvarania_M6.CMD.ErrorRESET:= FALSE;
    ELSIF CasResetServaZdvihuZvarania.Q THEN
        P2_Zvaranie.ServoZdvihuZvarania_M6.CMD.ErrorRESET:= FALSE;
    END_IF

    CasResetServaZdvihuZakladaca.PT:= T#2s;
    CasResetServaZdvihuZakladaca.IN:= P2_ZakladacTesnenia.ServoZdvihuZakladaca_M4.CMD.ErrorRESET;
    CasResetServaZdvihuZakladaca();

    CasResetServaPojazduZakladaca.PT:= T#2s;
    CasResetServaPojazduZakladaca.IN:= P2_ZakladacTesnenia.ServoPojazduVozika_M5.CMD.ErrorRESET;
    CasResetServaPojazduZakladaca();

    CasResetovaniaServaSrobovaniaOsX.PT:= T#2s;
    CasResetovaniaServaSrobovaniaOsX.IN:= P2_Srobovanie.ServoManipulOsX_M10.CMD.ErrorRESET;
    CasResetovaniaServaSrobovaniaOsX();

    CasResetovaniaServaSrobovaniaOsY.PT:= T#2s;
    CasResetovaniaServaSrobovaniaOsY.IN:= P2_Srobovanie.ServoManipulOsY_M9.CMD.ErrorRESET;
    CasResetovaniaServaSrobovaniaOsY();

    CasResetServaZdvihuZvarania.PT:= T#2s;
    CasResetServaZdvihuZvarania.IN:= P2_Zvaranie.ServoZdvihuZvarania_M6.CMD.ErrorRESET;
    CasResetServaZdvihuZvarania();

END_PROGRAM

PROGRAM _EXIT
	(* Insert code here *)

END_PROGRAM
```

#### Variables.var - Local variables
```iecst
VAR
	i : UINT;
	CasKontroly_TlakVzduchu : TON;
	CasKontroly_KAMsystem : TON;
	CasKontroly_Moduly : TON;
	CasKontroly_VentTerminalov : TON;
	CasKontroly_Skrutkovacky : TON;
	CasKontroly_Robota : TON;
	CasPoruchyServaZdvihuZakladaca : TON;
	CasPoruchyServaPojazduZakladaca : TON;
	CasPoruchyServaSrobovaniaOsX : TON;
	CasPoruchyServaSrobovaniaOsY : TON;
	CasPoruchyServaZdvihuZvarania : TON;
	CasResetServaZdvihuZakladaca : TON;
	CasResetServaPojazduZakladaca : TON;
	CasResetovaniaServaSrobovaniaOsX : TON;
	CasResetovaniaServaSrobovaniaOsY : TON;
	CasResetServaZdvihuZvarania : TON;
	a : INT;
END_VAR
```

### Program Logical/Alarmy/P34_Alarmy (IEC)
